Yaskawa INFORM job: TESTJOB1.JBI

/JOB
//NAME TESTJOB1
//POS
///NPOS 0,0,0,2,0,0
///TOOL 0
///POSTYPE PULSE
///PULSE
P00000=0,0,0,0,0,0
///USER 1
///POSTYPE USER
///RECTAN
///RCONF 0,0,0,0,0,0,0,0,0,0,0,0,0,0,0,0,0,0,0,0,0,0,0,0
P00003=300.000,0.000,0.000,0.0000,0.0000,0.0000
//INST
///DATE 2010/10/21 11:34
///ATTR SC,RW
///GROUP1 RB1
NOP
*LABEL
MOVL P000 V=83.3
MOVL P003 V=83.3
JUMP *LABEL
END
